// TIA Portal V15.1 export
// export: Created 2024-05-17T05:38:45.8173072Z, ExportSetting WithDefaults, DisplayName Totally Integrated Automation Portal, DisplayVersion V15.1 Update 5, DisplayName TIA Portal Openness, DisplayVersion V15.1 Update 5, DisplayName SINAMICS Startdrive Advanced, DisplayVersion V15.1, DisplayName G130, G150, S120, S150, SINAMICS MV, S210, DisplayVersion V15.1, DisplayName G110M, G120, G120C, G120D, G120P, DisplayVersion V15.1, DisplayName STEP 7 Professional, DisplayVersion V15.1 Update 5, DisplayName STEP 7 Safety, DisplayVersion V15.1, DisplayName WinCC Professional, DisplayVersion V15.1 Update 5, DisplayName SIMATIC Visualization Architect, DisplayVersion V15.1
FUNCTION_BLOCK "LGBGateLock-MGB-Maint"   // FB6628, FBD
TITLE = LGateLock-MGB / LGateLock-MGB-Maint
{ S7_Optimized_Access := 'TRUE' }
VERSION : 0.1
// =============================================================================
// This module is used for Euchner steered doorlock with 6 (lamp)pushbuttons and emergency stop
// Artikel 124573 MGB-L1HEB-PNA-R-124573
// Artikel 124575 MGB-L1HEB-PNA-L-124575
// 
// This module generates also a word containing all necessary information for HMI 
// Icon Animation, and a word with all information for HMI safety module 
// diagnostic screen. 
// =============================================================================
// stored: AutoNumber false, IsIECCheckEnabled false, IsRetainMemResEnabled false, MemoryReserve 100, SetENOAutomatically False, UDAEnableTagReadback false
   VAR_INPUT
      I_SafetyGateInput { ExternalAccessible := 'False'; ExternalVisible := 'False'; ExternalWritable := 'False'} : Bool;   // Input safety alarm (normally closed) / Input safety alarm (Summary door closed [T] and handle closed [R] - SK) / Input safety gate alarm (Summary door closed [T] and handle closed [R] - SK)
      I_Q { ExternalAccessible := 'False'; ExternalVisible := 'False'; ExternalWritable := 'False'} : Bool;   // Input safety alarm (normally closed) / Input Safety Alarm (normally closed) / Input Safety Logic Result Alarm (normally closed)
      I_EnableAlarm { ExternalAccessible := 'False'; ExternalVisible := 'False'; ExternalWritable := 'False'} : Bool := TRUE;   // Enable alarm from upper level
      I_StartPBInd { ExternalAccessible := 'False'; ExternalVisible := 'False'; ExternalWritable := 'False'} : Bool;   // Start PB indication
      I_AlarmResetPBInd { ExternalAccessible := 'False'; ExternalVisible := 'False'; ExternalWritable := 'False'} : Bool;   // Alarm reset PB indicatio / Alarm Reset PB Indication
      I_AccessStopReached { ExternalAccessible := 'False'; ExternalVisible := 'False'; ExternalWritable := 'False'} : Bool;   // Stop position reached for Request access / Access stop position reached
      I_CycleStopRequest { ExternalAccessible := 'False'; ExternalVisible := 'False'; ExternalWritable := 'False'} : Bool;   // Cycle stop request / Maintenance request
      I_CycleStopReached { ExternalAccessible := 'False'; ExternalVisible := 'False'; ExternalWritable := 'False'} : Bool;   // Cycle stop reached
      I_MaintRequest { ExternalAccessible := 'False'; ExternalVisible := 'False'; ExternalWritable := 'False'} : Bool;   // Cycle stop request / Maintenance request
      I_MaintReached { ExternalAccessible := 'False'; ExternalVisible := 'False'; ExternalWritable := 'False'} : Bool;   // Maintenance Position Reached
      I_SafetyCard_Pass_Out { ExternalAccessible := 'False'; ExternalVisible := 'False'; ExternalWritable := 'False'} : Bool;   // Passivation output
      I_SafetyCard_ACK_REQ { ExternalAccessible := 'False'; ExternalVisible := 'False'; ExternalWritable := 'False'} : Bool;   // ACK_REQ
      I_SafetyCard_ACK_DIAG { ExternalAccessible := 'False'; ExternalVisible := 'False'; ExternalWritable := 'False'} : Byte;   // ACK_DIAG
      "C_MGB-B" { ExternalAccessible := 'False'; ExternalVisible := 'False'; ExternalWritable := 'False'} : HW_SUBMODULE;   // Hw Config
      "C_MGB-EmergencySwitchStd" { ExternalAccessible := 'False'; ExternalVisible := 'False'; ExternalWritable := 'False'} : HW_SUBMODULE;   // Hw Config
      "C_MGB-L" { ExternalAccessible := 'False'; ExternalVisible := 'False'; ExternalWritable := 'False'} : HW_SUBMODULE;   // Hw Config
      "C_MBG-EnablingSwitchStd" { ExternalAccessible := 'False'; ExternalVisible := 'False'; ExternalWritable := 'False'} : HW_SUBMODULE;   // Hw Config
      "C_MBG-DIAG" { ExternalAccessible := 'False'; ExternalVisible := 'False'; ExternalWritable := 'False'} : HW_SUBMODULE;   // Hw Config
   END_VAR
   VAR_OUTPUT
      O_StartPB { ExternalAccessible := 'False'; ExternalVisible := 'False'; ExternalWritable := 'False'} : Bool;   // Pushbutton Start
      O_ResetAlarmPB { ExternalAccessible := 'False'; ExternalVisible := 'False'; ExternalWritable := 'False'} : Bool;   // Pushbutton Reset Alarm
      O_StopPB { ExternalAccessible := 'False'; ExternalVisible := 'False'; ExternalWritable := 'False'} : Bool;   // Pushbutton Stop (Delayed)
      O_EnablingSwitchPB { ExternalAccessible := 'False'; ExternalVisible := 'False'; ExternalWritable := 'False'} : Bool;   // Pushbutton Start / Pushbutton Enabling Switch
      "O_EnablingSwitch+PB" { ExternalAccessible := 'False'; ExternalVisible := 'False'; ExternalWritable := 'False'} : Bool;   // Pushbutton Start / Pushbutton Enabling Switch +
      "O_EnablingSwitch-PB" { ExternalAccessible := 'False'; ExternalVisible := 'False'; ExternalWritable := 'False'} : Bool;   // Pushbutton Start / Pushbutton Enabling Switch -
      O_MaintReq { ExternalAccessible := 'False'; ExternalVisible := 'False'; ExternalWritable := 'False'} : Bool;   // Switch Maintenance
      O_CycleStopReq { ExternalAccessible := 'False'; ExternalVisible := 'False'; ExternalWritable := 'False'} : Bool;   // Request for cycle stop / Request for Cycle Stop
      O_AccesStopReq { ExternalAccessible := 'False'; ExternalVisible := 'False'; ExternalWritable := 'False'} : Bool;   // Request for cycle stop / Request for Cycle Stop / Request for Acces Stop / Request for Access
      O_SafetyGateAlarm { ExternalAccessible := 'False'; ExternalVisible := 'False'; ExternalWritable := 'False'} : Bool;   // Alarm / Safety Alarm (Gate open) / Safety Gate Alarm
      O_EnablingSwitchAlarm { ExternalAccessible := 'False'; ExternalVisible := 'False'; ExternalWritable := 'False'} : Bool;   // Alarm / Enabling Switch Alarm (B) / Safety Gate Alarm
      O_SolenoidAlarm { ExternalAccessible := 'False'; ExternalVisible := 'False'; ExternalWritable := 'False'} : Bool;   // Summation Alarm A / Alarm / Alarm (C) / Solenoid Alarm
      O_AccessReqAlarm { ExternalAccessible := 'False'; ExternalVisible := 'False'; ExternalWritable := 'False'} : Bool;   // Alarm (C)
      O_MGBDiagWarning { ExternalAccessible := 'False'; ExternalVisible := 'False'; ExternalWritable := 'False'} : Bool;   // Summation Alarm C / Warning / Warning (D) / MGB diagnostic Warning
      O_AlarmABCondition { ExternalAccessible := 'False'; ExternalVisible := 'False'; ExternalWritable := 'False'} : Bool;   // Alarm AB Condition / Alarm AB condition
   END_VAR
   VAR_IN_OUT
      IO_Modes : "Modes";   // Modes
      H_HMI : "H_HMI";   // Animation
      "H_GateLock-MGB" : "H_GateLock-MGB-Maint";   // Animation
      C_AlarmHighSeverityA { ExternalAccessible := 'False'; ExternalVisible := 'False'; ExternalWritable := 'False'} : Bool := TRUE;   // Interlock alarm for Set direction / Alarm severity / Alarm severity A
      C_AlarmHighSeverityB { ExternalAccessible := 'False'; ExternalVisible := 'False'; ExternalWritable := 'False'} : Bool := False;   // Interlock alarm for Set direction / Alarm severity / Alarm severity B
      C_Warning { ExternalAccessible := 'False'; ExternalVisible := 'False'; ExternalWritable := 'False'} : Bool := False;   // Warning
   END_VAR
   VAR
      MGB { ExternalAccessible := 'False'; ExternalVisible := 'False'; ExternalWritable := 'False'} : "Euchner-MGB-Maint";   // UDT
      SafetyCard { ExternalAccessible := 'False'; ExternalVisible := 'False'; ExternalWritable := 'False'} : "SafetyCard";   // Safety Card UDT
      Pass_Out { ExternalAccessible := 'False'; ExternalVisible := 'False'; ExternalWritable := 'False'} : Bool;   // Acknowledgement request / Passivation output
      Ack_Req { ExternalAccessible := 'False'; ExternalVisible := 'False'; ExternalWritable := 'False'} : Bool;   // Acknowledgement request / Acknowledge Request
      Timeout_F_I_O { ExternalAccessible := 'False'; ExternalVisible := 'False'; ExternalWritable := 'False'} : Bool;   // Timeout detected by F-I/O
      ChannelFault_F_I_O { ExternalAccessible := 'False'; ExternalVisible := 'False'; ExternalWritable := 'False'} : Bool;   // F-I/O fault or channel fault detected by F-I/O
      CRCSeqError_F_I_O { ExternalAccessible := 'False'; ExternalVisible := 'False'; ExternalWritable := 'False'} : Bool;   // CRC error or sequence number error detected by F-I/O
      Timeout_F_Sys { ExternalAccessible := 'False'; ExternalVisible := 'False'; ExternalWritable := 'False'} : Bool;   // Timeout detected by F-System
      SeqError_F_Sys { ExternalAccessible := 'False'; ExternalVisible := 'False'; ExternalWritable := 'False'} : Bool;   // Sequence number error detected by F-system
      CRCError_F_Sys { ExternalAccessible := 'False'; ExternalVisible := 'False'; ExternalWritable := 'False'} : Bool;   // CRC error detected by F-system
      DelayStop { ExternalAccessible := 'False'; ExternalVisible := 'False'; ExternalWritable := 'False'} : Bool;   // Stop pushbutton delayed
      DelayMaint { ExternalAccessible := 'False'; ExternalVisible := 'False'; ExternalWritable := 'False'} : Bool;   // Maintenance pushbutton delayed
      SafetyGateAlarm { ExternalAccessible := 'False'; ExternalVisible := 'False'; ExternalWritable := 'False'} : Bool;   // Alarm / Safety Gate Alarm
      SafetyGateAlarmCond { ExternalAccessible := 'False'; ExternalVisible := 'False'; ExternalWritable := 'False'} : Bool;   // Alarm condition / Safety Gate Alarm condition
      EnablingSwitchAlarm { ExternalAccessible := 'False'; ExternalVisible := 'False'; ExternalWritable := 'False'} : Bool;   // Alarm / Safety Gate Alarm
      EnablingSwitchAlarmCond { ExternalAccessible := 'False'; ExternalVisible := 'False'; ExternalWritable := 'False'} : Bool;   // Alarm condition / Safety Gate Alarm condition
      SolenoidAlarm { ExternalAccessible := 'False'; ExternalVisible := 'False'; ExternalWritable := 'False'} : Bool;   // Alarm / Solenoid Alarm
      SolenoidAlarmCond { ExternalAccessible := 'False'; ExternalVisible := 'False'; ExternalWritable := 'False'} : Bool;   // Alarm condition / Solenoid Alarm condition
      AccessReqAlarm { ExternalAccessible := 'False'; ExternalVisible := 'False'; ExternalWritable := 'False'} : Bool;   // Alarm / Solenoid Alarm / Access Request Alarm
      DelayCheckGuardUnlocking { ExternalAccessible := 'False'; ExternalVisible := 'False'; ExternalWritable := 'False'} : Bool;   // Alarm / Alarm Delay to check guard locking / Alarm Delay to check guard unlocking
      AccessReqSel { ExternalAccessible := 'False'; ExternalVisible := 'False'; ExternalWritable := 'False'} : Bool;   // Request access memory / Request access selected
      AccessReq { ExternalAccessible := 'False'; ExternalVisible := 'False'; ExternalWritable := 'False'} : Bool;   // Request access memory / Request access
      NotAutoMem { ExternalAccessible := 'False'; ExternalVisible := 'False'; ExternalWritable := 'False'} : Bool;   // Pushbutton stop memory
      DelayTimerPbStop { ExternalAccessible := 'False'; ExternalVisible := 'False'; ExternalWritable := 'False'} : IEC_TIMER;   // Delay timer for Stop pushbutton
      DelayTimerSolenoidAlarm { ExternalAccessible := 'False'; ExternalVisible := 'False'; ExternalWritable := 'False'} : IEC_TIMER;   // Delay timer for solenoid Alarm
      DelayTimerMaintPb { ExternalAccessible := 'False'; ExternalVisible := 'False'; ExternalWritable := 'False'} : IEC_TIMER;   // Delay timer for maintenance pushbutton
      DelayOFFAutoMode { ExternalAccessible := 'False'; ExternalVisible := 'False'; ExternalWritable := 'False'} : IEC_TIMER;   // Delay OFF auto mode
      Edge { ExternalAccessible := 'False'; ExternalVisible := 'False'; ExternalWritable := 'False'} : Array[1..10] of Bool;   // Edges / Edge
      _ToggleReqAccess { ExternalAccessible := 'False'; ExternalVisible := 'False'; ExternalWritable := 'False'} : "LToggle";   // Toggle request access / Toggle access request
   END_VAR
   VAR_TEMP   // added for the SCL form of the ladder/FBD networks
      _w1 : Bool;
      _w2 : Bool;
   END_VAR
BEGIN

NETWORK
TITLE = **** 1 - Inputs **** Input Range - Output Range Euchner Safetylock
// Input Range - Output Range Euchner Safetylock
// Input range MGB-B
// Bit      7          6          5          4             3             2               1              0
// Byte 0   -          -          Stop       Cycle Stop    Maintenance   Request Access  Reset Alarm    Start

// Input range MGB-L
// Bit      7          6          5          4             3             2               1              0
// Byte 0   -          -          -          -             -             Door Locked     Handle Closed  Door Closed


// Output range MGB-B
// Bit      7          6          5          4             3             2               1              0
// Byte 0   -          -          -          Cycle Stop    Maintenance   Request Access  Reset Alarm    Start

// Output range MGB-L
// Bit      7          6          5          4             3             2               1              0
// Byte 0   -          -          -          -             -             -               -              Guard Locking



REGION Network 2: **** 1 - Inputs **** IN-Parameter reading and storing to local variables for MGB-B
   // IN-Parameter reading and storing to local variables for MGB-B
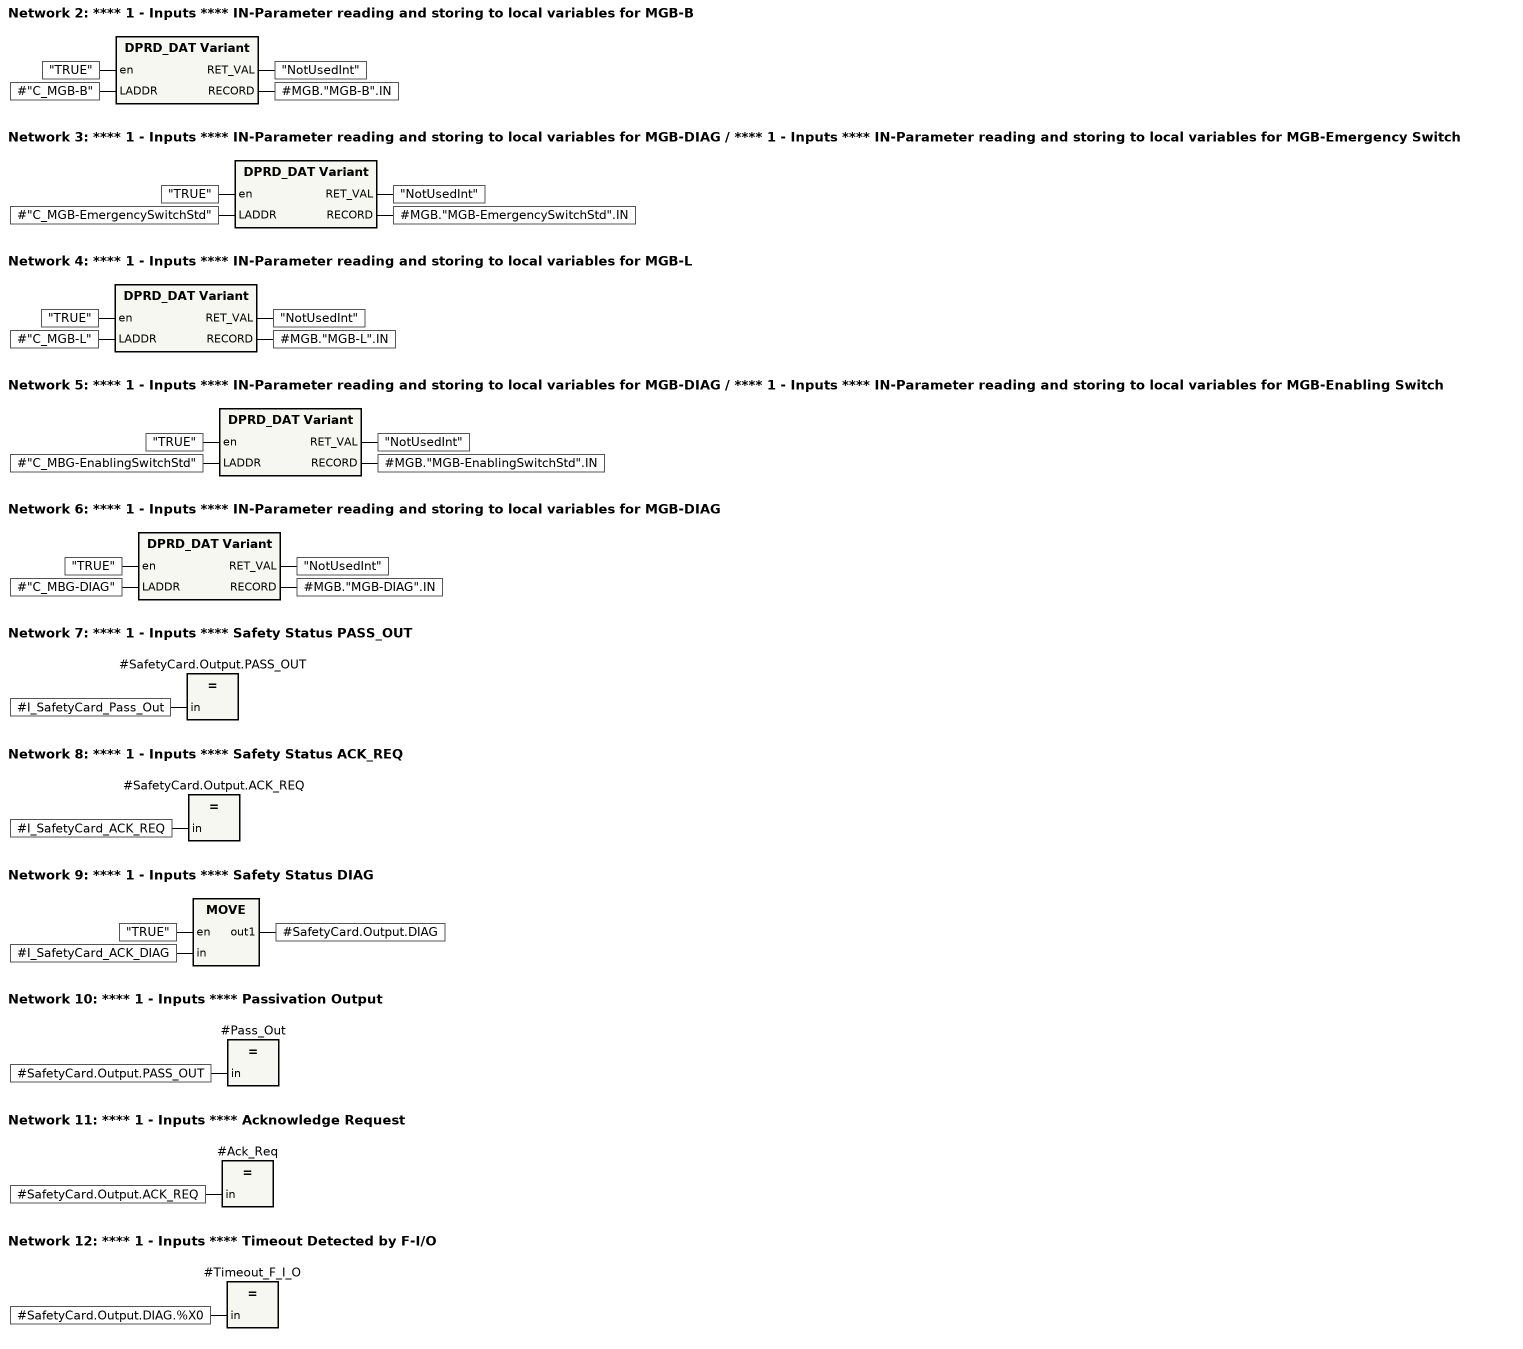
   IF "TRUE" THEN "NotUsedInt" := DPRD_DAT(LADDR := #"C_MGB-B", RECORD => #MGB."MGB-B".IN); END_IF;
END_REGION

REGION Network 3: **** 1 - Inputs **** IN-Parameter reading and storing to local variables for MGB-DIAG / **** 1 - Inputs **** IN-Parameter reading and storing to local variables for MGB-Emergency Switch
   // IN-Parameter reading and storing to local variables for MGB-DIAG / IN-Parameter reading and storing to local variables for MGB-Emergency Switch
   IF "TRUE" THEN
       "NotUsedInt" := DPRD_DAT(LADDR := #"C_MGB-EmergencySwitchStd", RECORD => #MGB."MGB-EmergencySwitchStd".IN);
   END_IF;
END_REGION

REGION Network 4: **** 1 - Inputs **** IN-Parameter reading and storing to local variables for MGB-L
   // IN-Parameter reading and storing to local variables for MGB-L
   IF "TRUE" THEN "NotUsedInt" := DPRD_DAT(LADDR := #"C_MGB-L", RECORD => #MGB."MGB-L".IN); END_IF;
END_REGION

REGION Network 5: **** 1 - Inputs **** IN-Parameter reading and storing to local variables for MGB-DIAG / **** 1 - Inputs **** IN-Parameter reading and storing to local variables for MGB-Enabling Switch
   // IN-Parameter reading and storing to local variables for MGB-DIAG / IN-Parameter reading and storing to local variables for MGB-Enabling Switch
   IF "TRUE" THEN
       "NotUsedInt" := DPRD_DAT(LADDR := #"C_MBG-EnablingSwitchStd", RECORD => #MGB."MGB-EnablingSwitchStd".IN);
   END_IF;
END_REGION

REGION Network 6: **** 1 - Inputs **** IN-Parameter reading and storing to local variables for MGB-DIAG
   // IN-Parameter reading and storing to local variables for MGB-DIAG
   IF "TRUE" THEN "NotUsedInt" := DPRD_DAT(LADDR := #"C_MBG-DIAG", RECORD => #MGB."MGB-DIAG".IN); END_IF;
END_REGION

REGION Network 7: **** 1 - Inputs **** Safety Status PASS_OUT
   // Safety Status PASS_OUT
   #SafetyCard.Output.PASS_OUT := #I_SafetyCard_Pass_Out;
END_REGION

REGION Network 8: **** 1 - Inputs **** Safety Status ACK_REQ
   // Safety Status ACK_REQ
   #SafetyCard.Output.ACK_REQ := #I_SafetyCard_ACK_REQ;
END_REGION

REGION Network 9: **** 1 - Inputs **** Safety Status DIAG
   // Safety Status DIAG
   IF "TRUE" THEN #SafetyCard.Output.DIAG := #I_SafetyCard_ACK_DIAG; END_IF;
END_REGION

REGION Network 10: **** 1 - Inputs **** Passivation Output
   // Passivation Output
   #Pass_Out := #SafetyCard.Output.PASS_OUT;
END_REGION

REGION Network 11: **** 1 - Inputs **** Acknowledge Request
   // Acknowledge Request
   #Ack_Req := #SafetyCard.Output.ACK_REQ;
END_REGION

REGION Network 12: **** 1 - Inputs **** Timeout Detected by F-I/O
   // ### Timeout Detected by F-I/O - must be checked
   #Timeout_F_I_O := #SafetyCard.Output.DIAG.%X0;
END_REGION

REGION Network 13: **** 1 - Inputs **** F-I/O fault or Channel Fault Detected by F-I/O
   // F-I/O fault or Channel Fault Detected by F-I/O
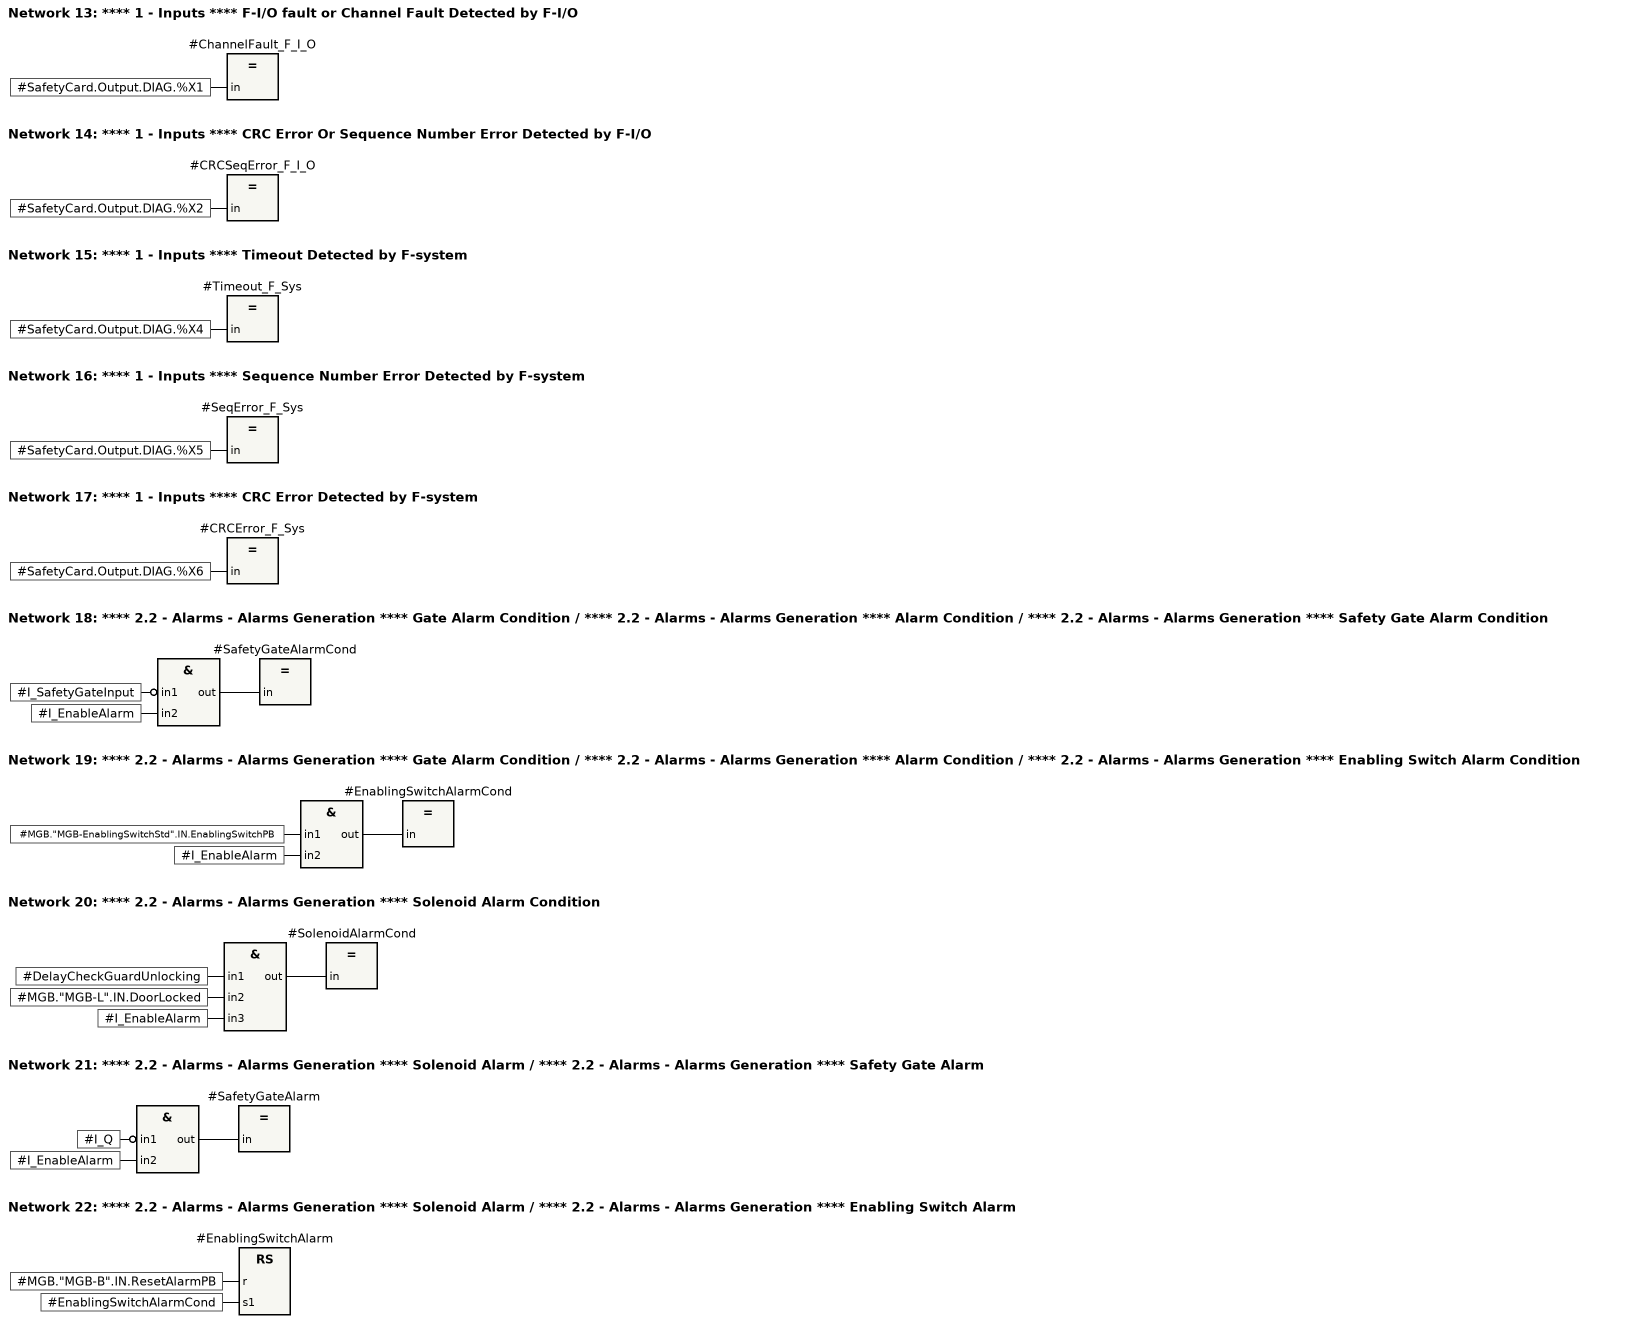
   #ChannelFault_F_I_O := #SafetyCard.Output.DIAG.%X1;
END_REGION

REGION Network 14: **** 1 - Inputs **** CRC Error Or Sequence Number Error Detected by F-I/O
   // CRC Error Or Sequence Number Error Detected by F-I/O
   #CRCSeqError_F_I_O := #SafetyCard.Output.DIAG.%X2;
END_REGION

REGION Network 15: **** 1 - Inputs **** Timeout Detected by F-system
   // Timeout Detected by F-system
   #Timeout_F_Sys := #SafetyCard.Output.DIAG.%X4;
END_REGION

REGION Network 16: **** 1 - Inputs **** Sequence Number Error Detected by F-system
   // Sequence Number Error Detected by F-system
   #SeqError_F_Sys := #SafetyCard.Output.DIAG.%X5;
END_REGION

REGION Network 17: **** 1 - Inputs **** CRC Error Detected by F-system
   // CRC Error Detected by F-system
   #CRCError_F_Sys := #SafetyCard.Output.DIAG.%X6;
END_REGION

REGION Network 18: **** 2.2 - Alarms - Alarms Generation **** Gate Alarm Condition / **** 2.2 - Alarms - Alarms Generation **** Alarm Condition / **** 2.2 - Alarms - Alarms Generation **** Safety Gate Alarm Condition
   // Condition of the Gate Alarm for the Normal Closed input / Condition of the Safety Alarm for the Normal Closed input
   #SafetyGateAlarmCond := NOT #I_SafetyGateInput AND #I_EnableAlarm;
END_REGION

REGION Network 19: **** 2.2 - Alarms - Alarms Generation **** Gate Alarm Condition / **** 2.2 - Alarms - Alarms Generation **** Alarm Condition / **** 2.2 - Alarms - Alarms Generation **** Enabling Switch Alarm Condition
   // Condition of the Gate Alarm for the Normal Closed input / Condition of the Safety Alarm for the Normal Closed input / Condition of the Enabling Switch actiavted alarm
   #EnablingSwitchAlarmCond := #MGB."MGB-EnablingSwitchStd".IN.EnablingSwitchPB AND #I_EnableAlarm;
END_REGION

REGION Network 20: **** 2.2 - Alarms - Alarms Generation **** Solenoid Alarm Condition
   // Condition of guardlocking on and solenoid not activated
   #SolenoidAlarmCond := #DelayCheckGuardUnlocking AND #MGB."MGB-L".IN.DoorLocked AND #I_EnableAlarm;
END_REGION

REGION Network 21: **** 2.2 - Alarms - Alarms Generation **** Solenoid Alarm / **** 2.2 - Alarms - Alarms Generation **** Safety Gate Alarm
   // Solenoid alarm / Condition of the Safety Alarm for the Normal Closed input
   #SafetyGateAlarm := NOT #I_Q AND #I_EnableAlarm;
END_REGION

REGION Network 22: **** 2.2 - Alarms - Alarms Generation **** Solenoid Alarm / **** 2.2 - Alarms - Alarms Generation **** Enabling Switch Alarm
   // Solenoid alarm / Enabling Switch alarm
   IF #MGB."MGB-B".IN.ResetAlarmPB THEN
       #EnablingSwitchAlarm := FALSE;   // RS flip-flop
   END_IF;
   IF #EnablingSwitchAlarmCond THEN #EnablingSwitchAlarm := TRUE; END_IF;
END_REGION

REGION Network 23: **** 2.2 - Alarms - Alarms Generation **** Solenoid Alarm
   // Solenoid alarm
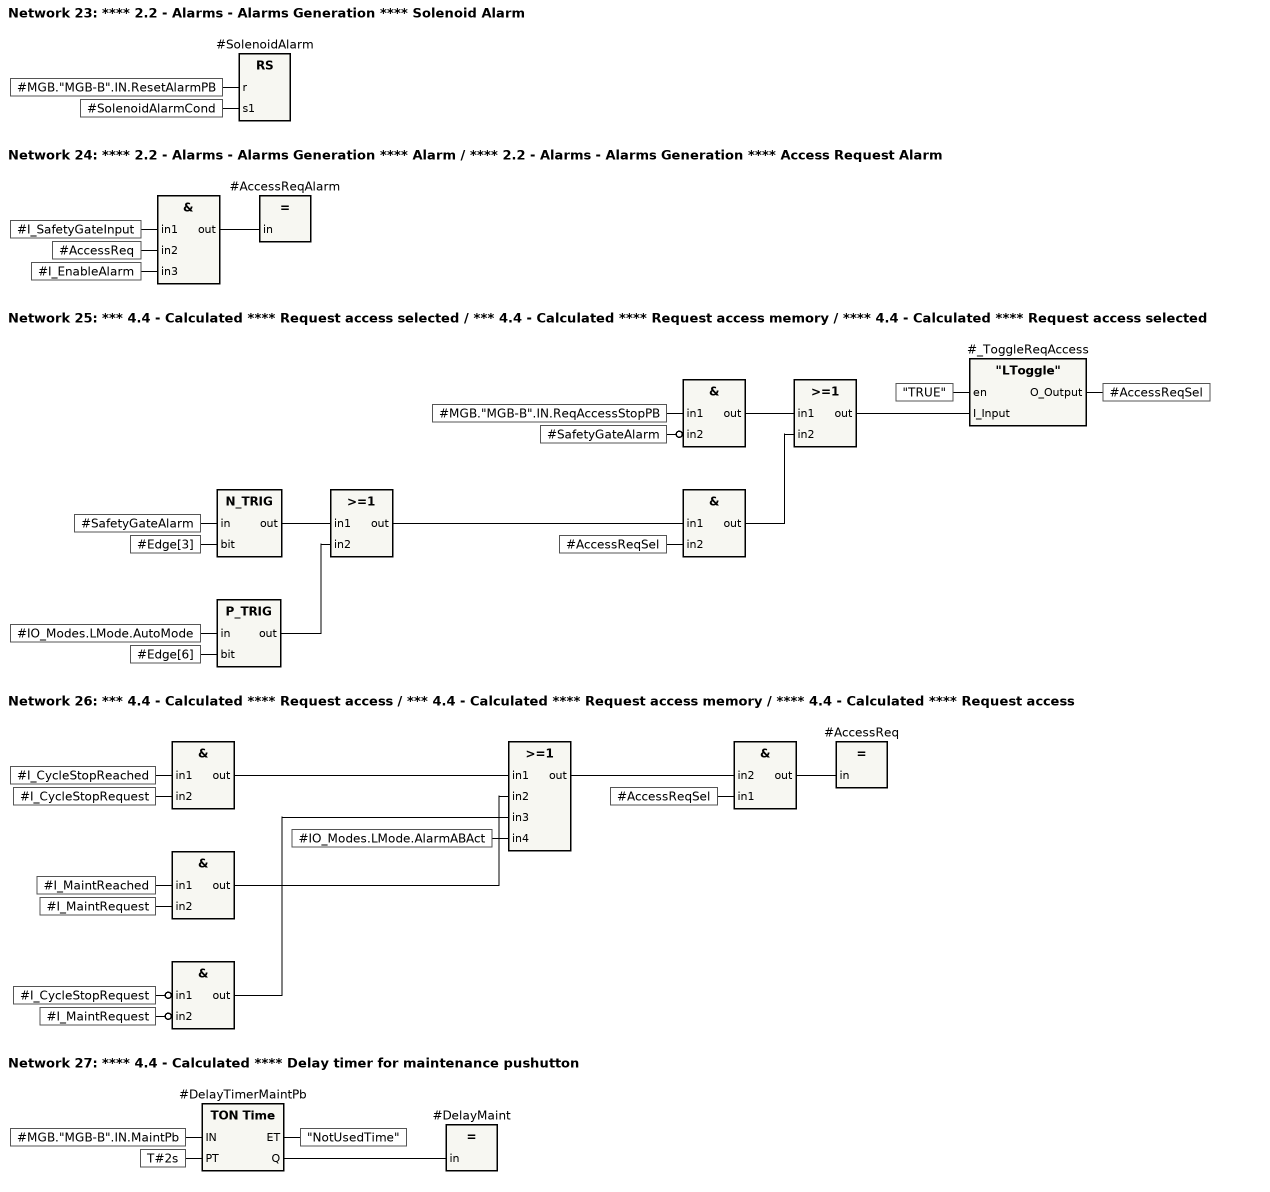
   IF #MGB."MGB-B".IN.ResetAlarmPB THEN
       #SolenoidAlarm := FALSE;   // RS flip-flop
   END_IF;
   IF #SolenoidAlarmCond THEN #SolenoidAlarm := TRUE; END_IF;
END_REGION

REGION Network 24: **** 2.2 - Alarms - Alarms Generation **** Alarm / **** 2.2 - Alarms - Alarms Generation **** Access Request Alarm
   // Creation of the Safety Alarm for the Normal Closed input / Alarm to notify that an access to the line is requested at the gate
   #AccessReqAlarm := #I_SafetyGateInput AND #AccessReq AND #I_EnableAlarm;
END_REGION

REGION Network 25: *** 4.4 - Calculated **** Request access selected / *** 4.4 - Calculated **** Request access memory / **** 4.4 - Calculated **** Request access selected
   // Request access selected / Request access memory
   #_w1 := NOT #SafetyGateAlarm AND #Edge[3];   // falling edge
   #Edge[3] := #SafetyGateAlarm;
   #_w2 := #IO_Modes.LMode.AutoMode AND NOT #Edge[6];   // rising edge
   #Edge[6] := #IO_Modes.LMode.AutoMode;
   IF "TRUE" THEN
       #_ToggleReqAccess(I_Input := (#MGB."MGB-B".IN.ReqAccessStopPB AND NOT #SafetyGateAlarm) OR ((#_w1 OR #_w2) AND #AccessReqSel),   // "LToggle"
                         O_Output => #AccessReqSel);
   END_IF;
END_REGION

REGION Network 26: *** 4.4 - Calculated **** Request access / *** 4.4 - Calculated **** Request access memory / **** 4.4 - Calculated **** Request access
   // Request access / Request access memory
   #AccessReq := ((#I_CycleStopReached AND #I_CycleStopRequest) OR (#I_MaintReached AND #I_MaintRequest) OR (NOT #I_CycleStopRequest AND NOT #I_MaintRequest) OR #IO_Modes.LMode.AlarmABAct) AND #AccessReqSel;
END_REGION

REGION Network 27: **** 4.4 - Calculated **** Delay timer for maintenance pushutton
   // Delay timer for maintenance pushutton
   #DelayTimerMaintPb.TON(IN := #MGB."MGB-B".IN.MaintPb, PT := T#2s, ET => "NotUsedTime");
   #DelayMaint := #DelayTimerMaintPb.Q;
END_REGION

REGION Network 28: *** 4.4 - Calculated **** Guard locking solenoid / **** 4.4 - Calculated **** Guard locking solenoid
   // Guard Locking Solenoid, Power to unlock (True = unlocked / False = locked) / Guard Locking Solenoid (True = locked / False = unlocked)
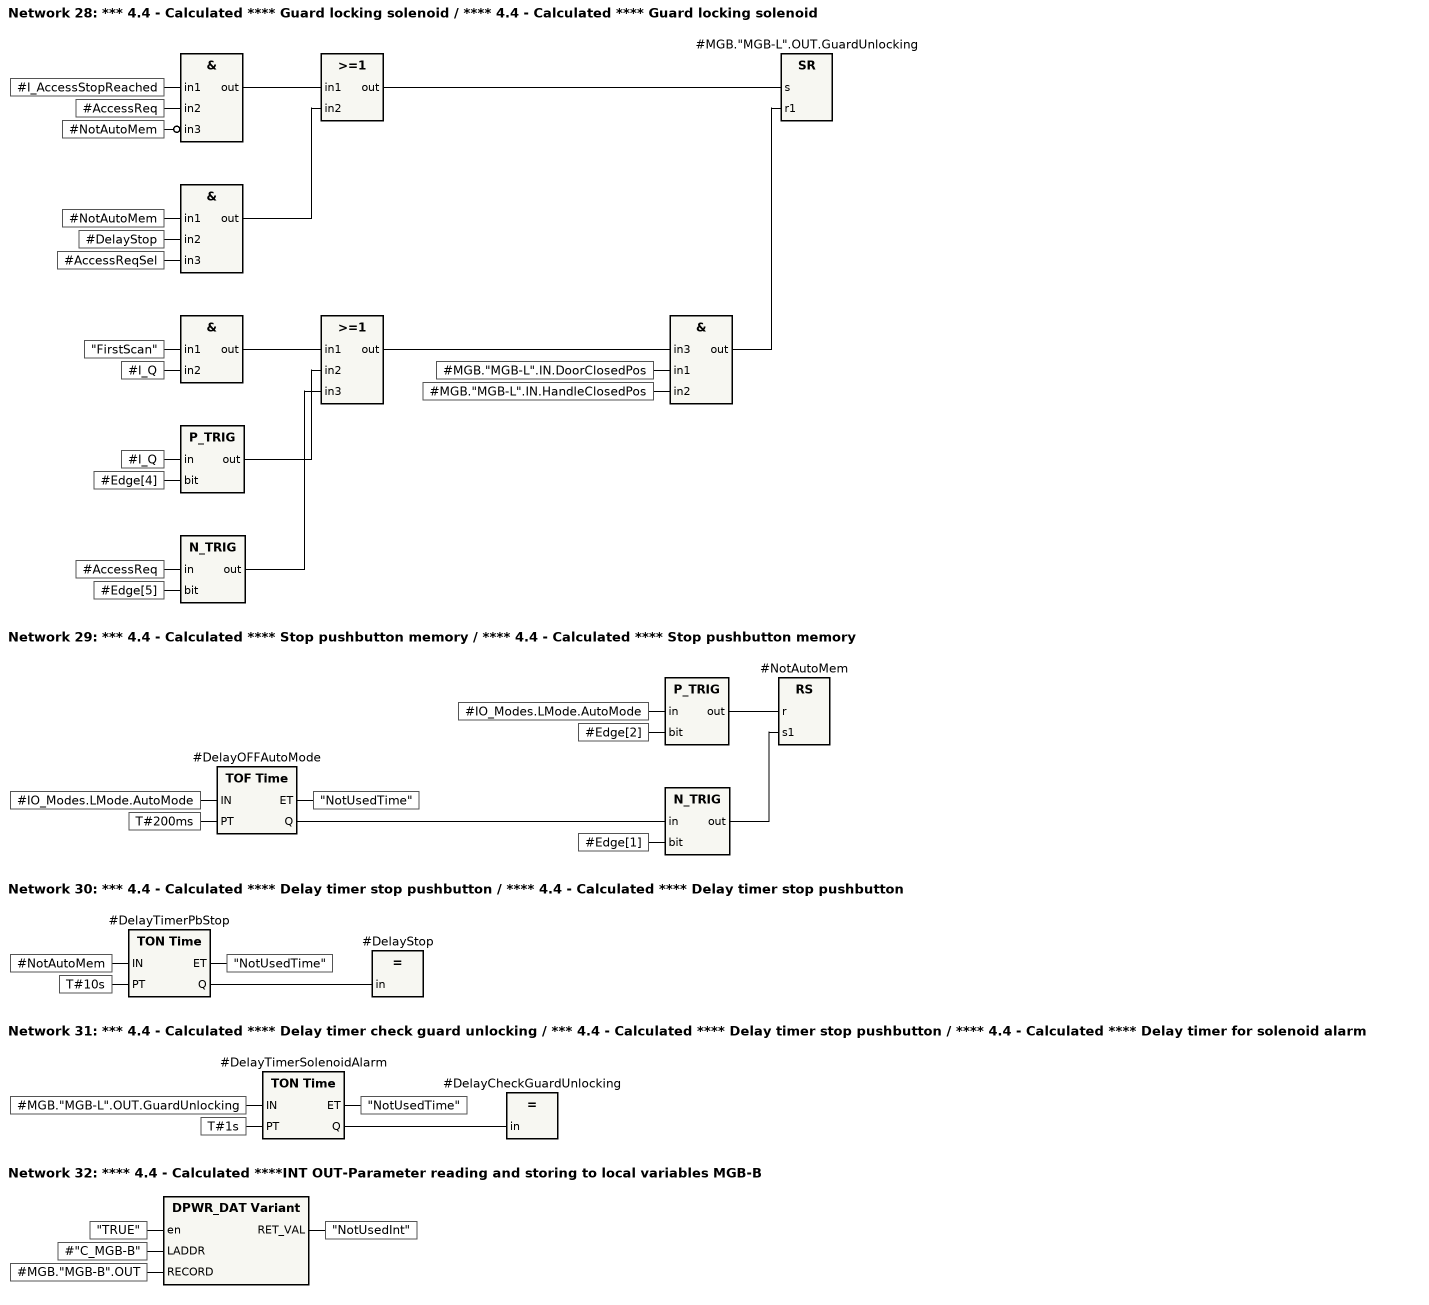
   #_w1 := #I_Q AND NOT #Edge[4];   // rising edge
   #Edge[4] := #I_Q;
   #_w2 := NOT #AccessReq AND #Edge[5];   // falling edge
   #Edge[5] := #AccessReq;
   IF (#I_AccessStopReached AND #AccessReq AND NOT #NotAutoMem) OR (#NotAutoMem AND #DelayStop AND #AccessReqSel) THEN
       #MGB."MGB-L".OUT.GuardUnlocking := TRUE;   // SR flip-flop
   END_IF;
   IF (("FirstScan" AND #I_Q) OR #_w1 OR #_w2) AND #MGB."MGB-L".IN.DoorClosedPos AND #MGB."MGB-L".IN.HandleClosedPos THEN
       #MGB."MGB-L".OUT.GuardUnlocking := FALSE;
   END_IF;
END_REGION

REGION Network 29: *** 4.4 - Calculated **** Stop pushbutton memory / **** 4.4 - Calculated **** Stop pushbutton memory
   // Stop pushbutton memory
   #_w1 := #IO_Modes.LMode.AutoMode AND NOT #Edge[2];   // rising edge
   #Edge[2] := #IO_Modes.LMode.AutoMode;
   #DelayOFFAutoMode.TOF(IN := #IO_Modes.LMode.AutoMode, PT := T#200ms, ET => "NotUsedTime");
   #_w2 := NOT #DelayOFFAutoMode.Q AND #Edge[1];   // falling edge
   #Edge[1] := #DelayOFFAutoMode.Q;
   IF #_w1 THEN
       #NotAutoMem := FALSE;   // RS flip-flop
   END_IF;
   IF #_w2 THEN #NotAutoMem := TRUE; END_IF;
END_REGION

REGION Network 30: *** 4.4 - Calculated **** Delay timer stop pushbutton / **** 4.4 - Calculated **** Delay timer stop pushbutton
   // Delay for Stop pushbutton
   #DelayTimerPbStop.TON(IN := #NotAutoMem, PT := T#10s, ET => "NotUsedTime");
   #DelayStop := #DelayTimerPbStop.Q;
END_REGION

REGION Network 31: *** 4.4 - Calculated **** Delay timer check guard unlocking / *** 4.4 - Calculated **** Delay timer stop pushbutton / **** 4.4 - Calculated **** Delay timer for solenoid alarm
   // Delay for checking of guard unlocking / Delay for Stop pushbutton / Delay timer for solenoid alarm
   #DelayTimerSolenoidAlarm.TON(IN := #MGB."MGB-L".OUT.GuardUnlocking, PT := T#1s, ET => "NotUsedTime");
   #DelayCheckGuardUnlocking := #DelayTimerSolenoidAlarm.Q;
END_REGION

REGION Network 32: **** 4.4 - Calculated ****INT OUT-Parameter reading and storing to local variables MGB-B
   // INT OUT-Parameter reading and storing to local variables MGB-B
   IF "TRUE" THEN "NotUsedInt" := DPWR_DAT(LADDR := #"C_MGB-B", RECORD := #MGB."MGB-B".OUT); END_IF;
END_REGION

REGION Network 33: **** 4.4 - Calculated ****INT OUT-Parameter reading and storing to local variables MGB Diag / **** 4.4 - Calculated ****INT OUT-Parameter reading and storing to local variables MGB-Emergency Switch
   // INT OUT-Parameter reading and storing to local variables MGB Diag / INT OUT-Parameter reading and storing to local variables MGB-Emergency Switch
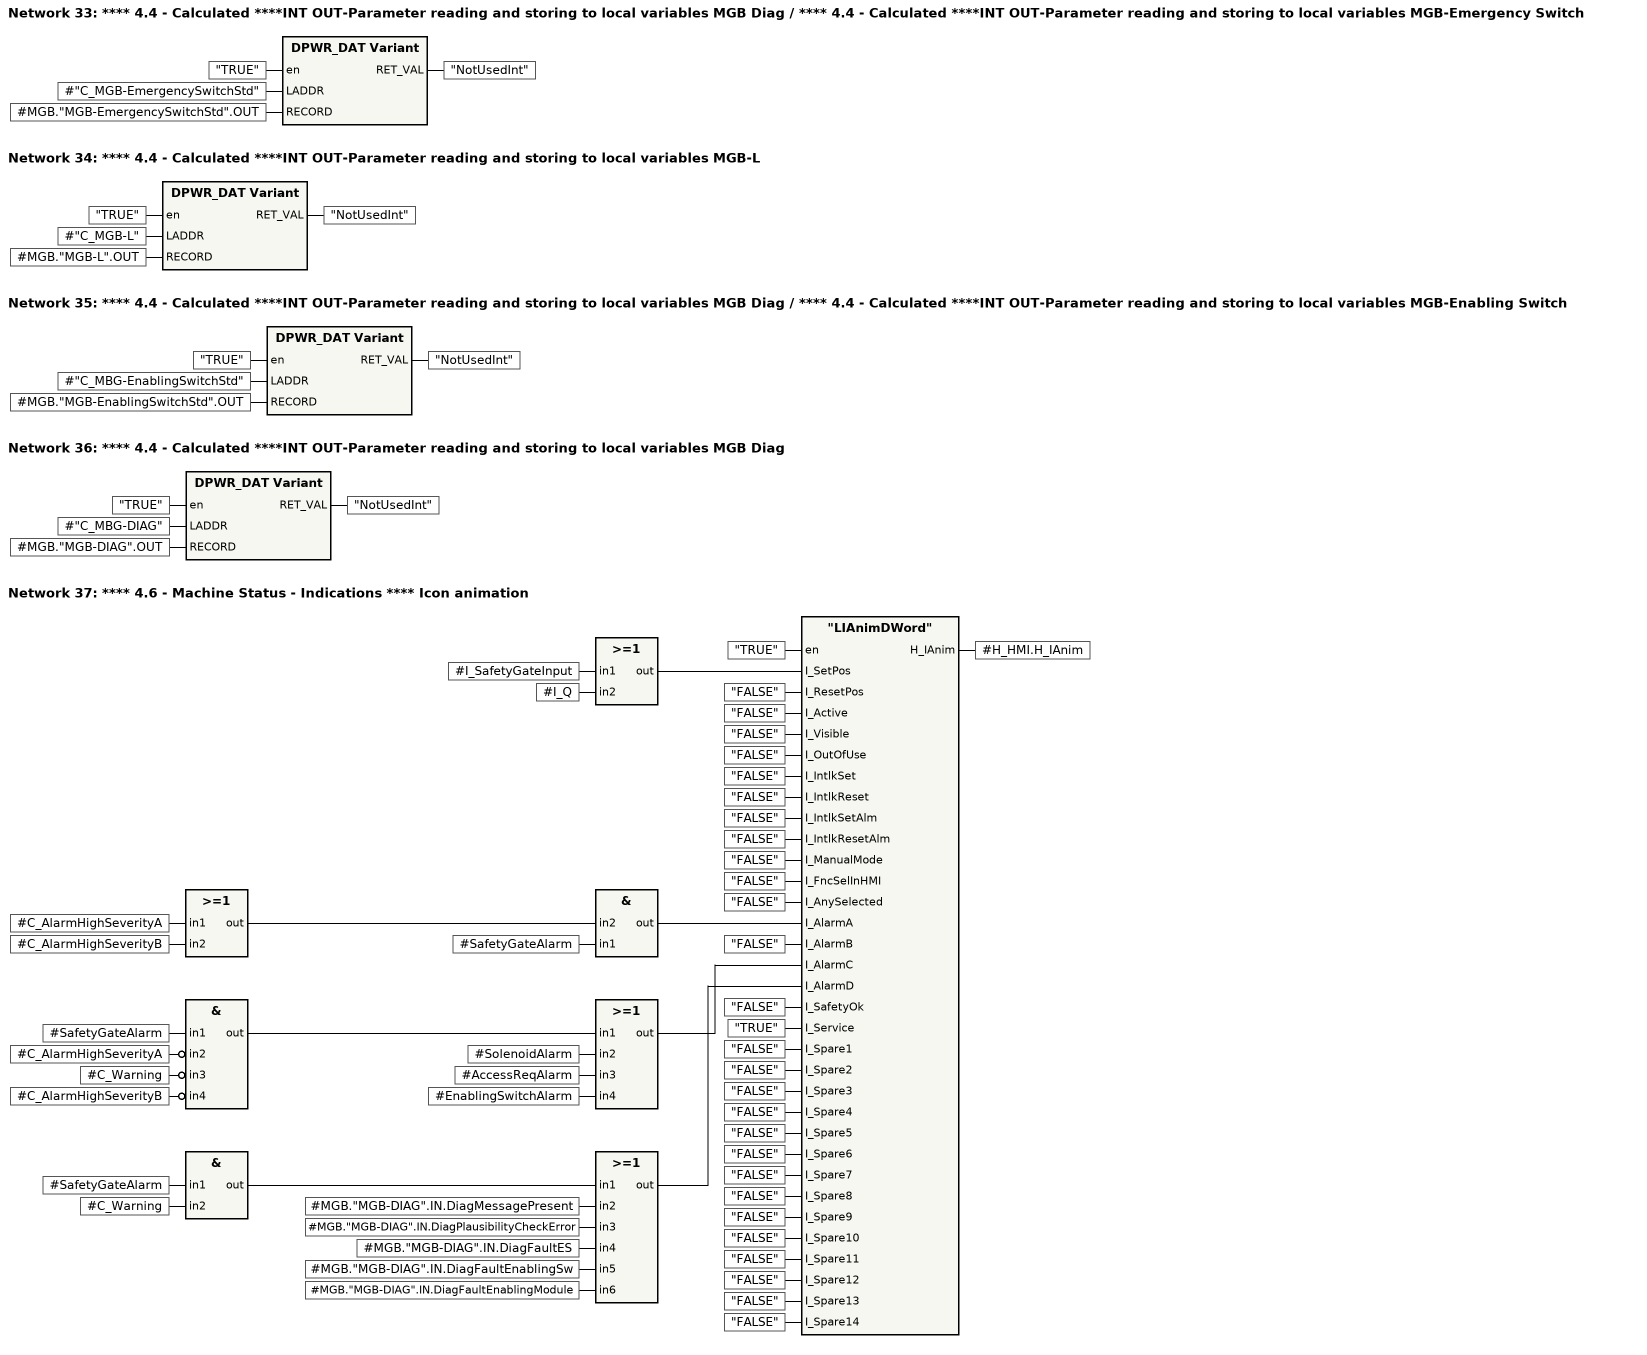
   IF "TRUE" THEN
       "NotUsedInt" := DPWR_DAT(LADDR := #"C_MGB-EmergencySwitchStd", RECORD := #MGB."MGB-EmergencySwitchStd".OUT);
   END_IF;
END_REGION

REGION Network 34: **** 4.4 - Calculated ****INT OUT-Parameter reading and storing to local variables MGB-L
   // INT OUT-Parameter reading and storing to local variables MGB-L
   IF "TRUE" THEN "NotUsedInt" := DPWR_DAT(LADDR := #"C_MGB-L", RECORD := #MGB."MGB-L".OUT); END_IF;
END_REGION

REGION Network 35: **** 4.4 - Calculated ****INT OUT-Parameter reading and storing to local variables MGB Diag / **** 4.4 - Calculated ****INT OUT-Parameter reading and storing to local variables MGB-Enabling Switch
   // INT OUT-Parameter reading and storing to local variables MGB Diag / INT OUT-Parameter reading and storing to local variables MGB-Enabling Switch
   IF "TRUE" THEN
       "NotUsedInt" := DPWR_DAT(LADDR := #"C_MBG-EnablingSwitchStd", RECORD := #MGB."MGB-EnablingSwitchStd".OUT);
   END_IF;
END_REGION

REGION Network 36: **** 4.4 - Calculated ****INT OUT-Parameter reading and storing to local variables MGB Diag
   // INT OUT-Parameter reading and storing to local variables MGB Diag
   IF "TRUE" THEN "NotUsedInt" := DPWR_DAT(LADDR := #"C_MBG-DIAG", RECORD := #MGB."MGB-DIAG".OUT); END_IF;
END_REGION

REGION Network 37: **** 4.6 - Machine Status - Indications **** Icon animation
   // Icon Animation
   IF "TRUE" THEN
       "LIAnimDWord"(I_SetPos := #I_SafetyGateInput OR #I_Q,
                     I_ResetPos := "FALSE",
                     I_Active := "FALSE",
                     I_Visible := "FALSE",
                     I_OutOfUse := "FALSE",
                     I_IntlkSet := "FALSE",
                     I_IntlkReset := "FALSE",
                     I_IntlkSetAlm := "FALSE",
                     I_IntlkResetAlm := "FALSE",
                     I_ManualMode := "FALSE",
                     I_FncSelInHMI := "FALSE",
                     I_AnySelected := "FALSE",
                     I_AlarmA := (#C_AlarmHighSeverityA OR #C_AlarmHighSeverityB) AND #SafetyGateAlarm,
                     I_AlarmB := "FALSE",
                     I_AlarmC := (#SafetyGateAlarm AND NOT #C_AlarmHighSeverityA AND NOT #C_Warning AND NOT #C_AlarmHighSeverityB) OR #SolenoidAlarm OR #AccessReqAlarm OR #EnablingSwitchAlarm,
                     I_AlarmD := (#SafetyGateAlarm AND #C_Warning) OR #MGB."MGB-DIAG".IN.DiagMessagePresent OR #MGB."MGB-DIAG".IN.DiagPlausibilityCheckError OR #MGB."MGB-DIAG".IN.DiagFaultES OR #MGB."MGB-DIAG".IN.DiagFaultEnablingSw OR #MGB."MGB-DIAG".IN.DiagFaultEnablingModule,
                     I_SafetyOk := "FALSE",
                     I_Service := "TRUE",
                     I_Spare1 := "FALSE",
                     I_Spare2 := "FALSE",
                     I_Spare3 := "FALSE",
                     I_Spare4 := "FALSE",
                     I_Spare5 := "FALSE",
                     I_Spare6 := "FALSE",
                     I_Spare7 := "FALSE",
                     I_Spare8 := "FALSE",
                     I_Spare9 := "FALSE",
                     I_Spare10 := "FALSE",
                     I_Spare11 := "FALSE",
                     I_Spare12 := "FALSE",
                     I_Spare13 := "FALSE",
                     I_Spare14 := "FALSE",
                     H_IAnim => #H_HMI.H_IAnim);
   END_IF;
END_REGION

REGION Network 38: **** 4.6 - Machine Status - Indications **** Animation
   // Animation
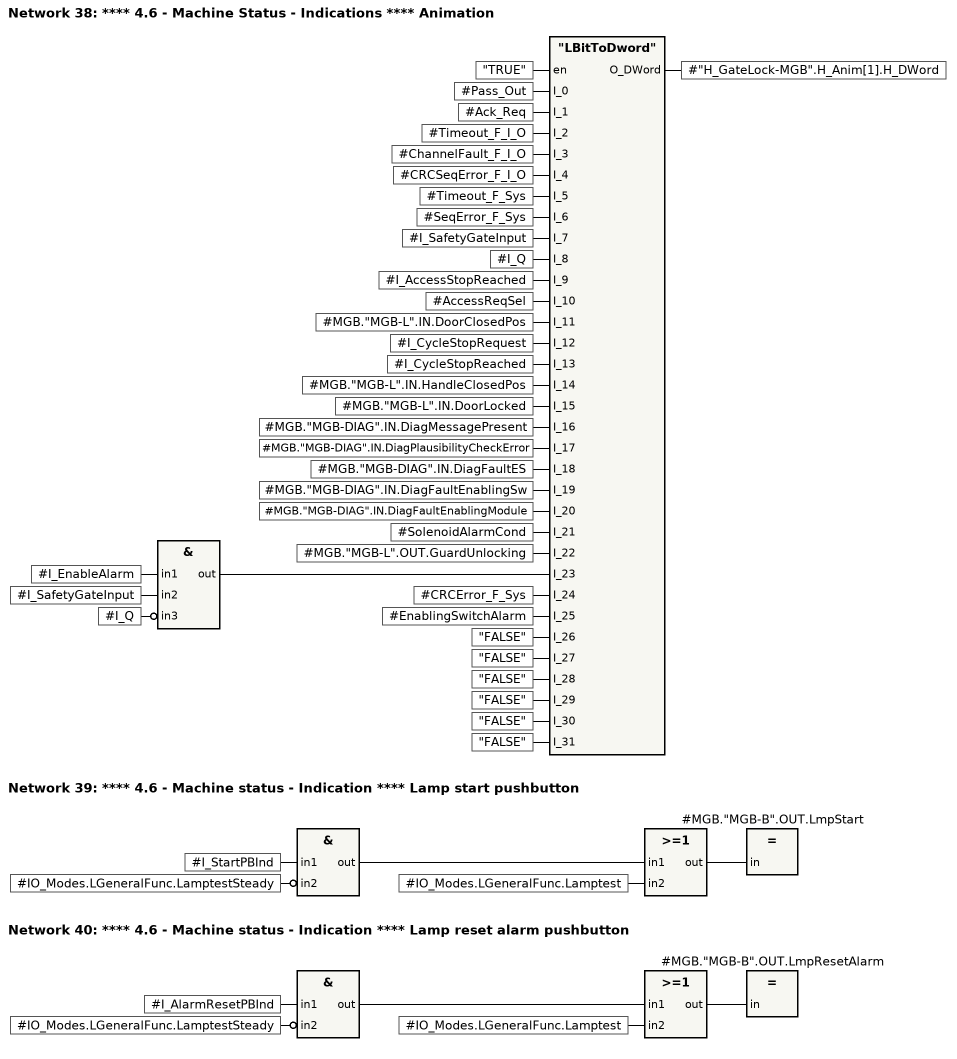
   IF "TRUE" THEN
       "LBitToDword"(I_0 := #Pass_Out,
                     I_1 := #Ack_Req,
                     I_2 := #Timeout_F_I_O,
                     I_3 := #ChannelFault_F_I_O,
                     I_4 := #CRCSeqError_F_I_O,
                     I_5 := #Timeout_F_Sys,
                     I_6 := #SeqError_F_Sys,
                     I_7 := #I_SafetyGateInput,
                     I_8 := #I_Q,
                     I_9 := #I_AccessStopReached,
                     I_10 := #AccessReqSel,
                     I_11 := #MGB."MGB-L".IN.DoorClosedPos,
                     I_12 := #I_CycleStopRequest,
                     I_13 := #I_CycleStopReached,
                     I_14 := #MGB."MGB-L".IN.HandleClosedPos,
                     I_15 := #MGB."MGB-L".IN.DoorLocked,
                     I_16 := #MGB."MGB-DIAG".IN.DiagMessagePresent,
                     I_17 := #MGB."MGB-DIAG".IN.DiagPlausibilityCheckError,
                     I_18 := #MGB."MGB-DIAG".IN.DiagFaultES,
                     I_19 := #MGB."MGB-DIAG".IN.DiagFaultEnablingSw,
                     I_20 := #MGB."MGB-DIAG".IN.DiagFaultEnablingModule,
                     I_21 := #SolenoidAlarmCond,
                     I_22 := #MGB."MGB-L".OUT.GuardUnlocking,
                     I_23 := #I_EnableAlarm AND #I_SafetyGateInput AND NOT #I_Q,
                     I_24 := #CRCError_F_Sys,
                     I_25 := #EnablingSwitchAlarm,
                     I_26 := "FALSE",
                     I_27 := "FALSE",
                     I_28 := "FALSE",
                     I_29 := "FALSE",
                     I_30 := "FALSE",
                     I_31 := "FALSE",
                     O_DWord => #"H_GateLock-MGB".H_Anim[1].H_DWord);
   END_IF;
END_REGION

REGION Network 39: **** 4.6 - Machine status - Indication **** Lamp start pushbutton
   // Start PB indication
   #MGB."MGB-B".OUT.LmpStart := (#I_StartPBInd AND NOT #IO_Modes.LGeneralFunc.LamptestSteady) OR #IO_Modes.LGeneralFunc.Lamptest;
END_REGION

REGION Network 40: **** 4.6 - Machine status - Indication **** Lamp reset alarm pushbutton
   // Reset Alarm PB indication / Alarm Reset PB indication
   #MGB."MGB-B".OUT.LmpResetAlarm := (#I_AlarmResetPBInd AND NOT #IO_Modes.LGeneralFunc.LamptestSteady) OR #IO_Modes.LGeneralFunc.Lamptest;
END_REGION

REGION Network 41: **** 4.6 - Machine status - Indication **** Lamp request access pushbutton
   // Request Acces PB indication
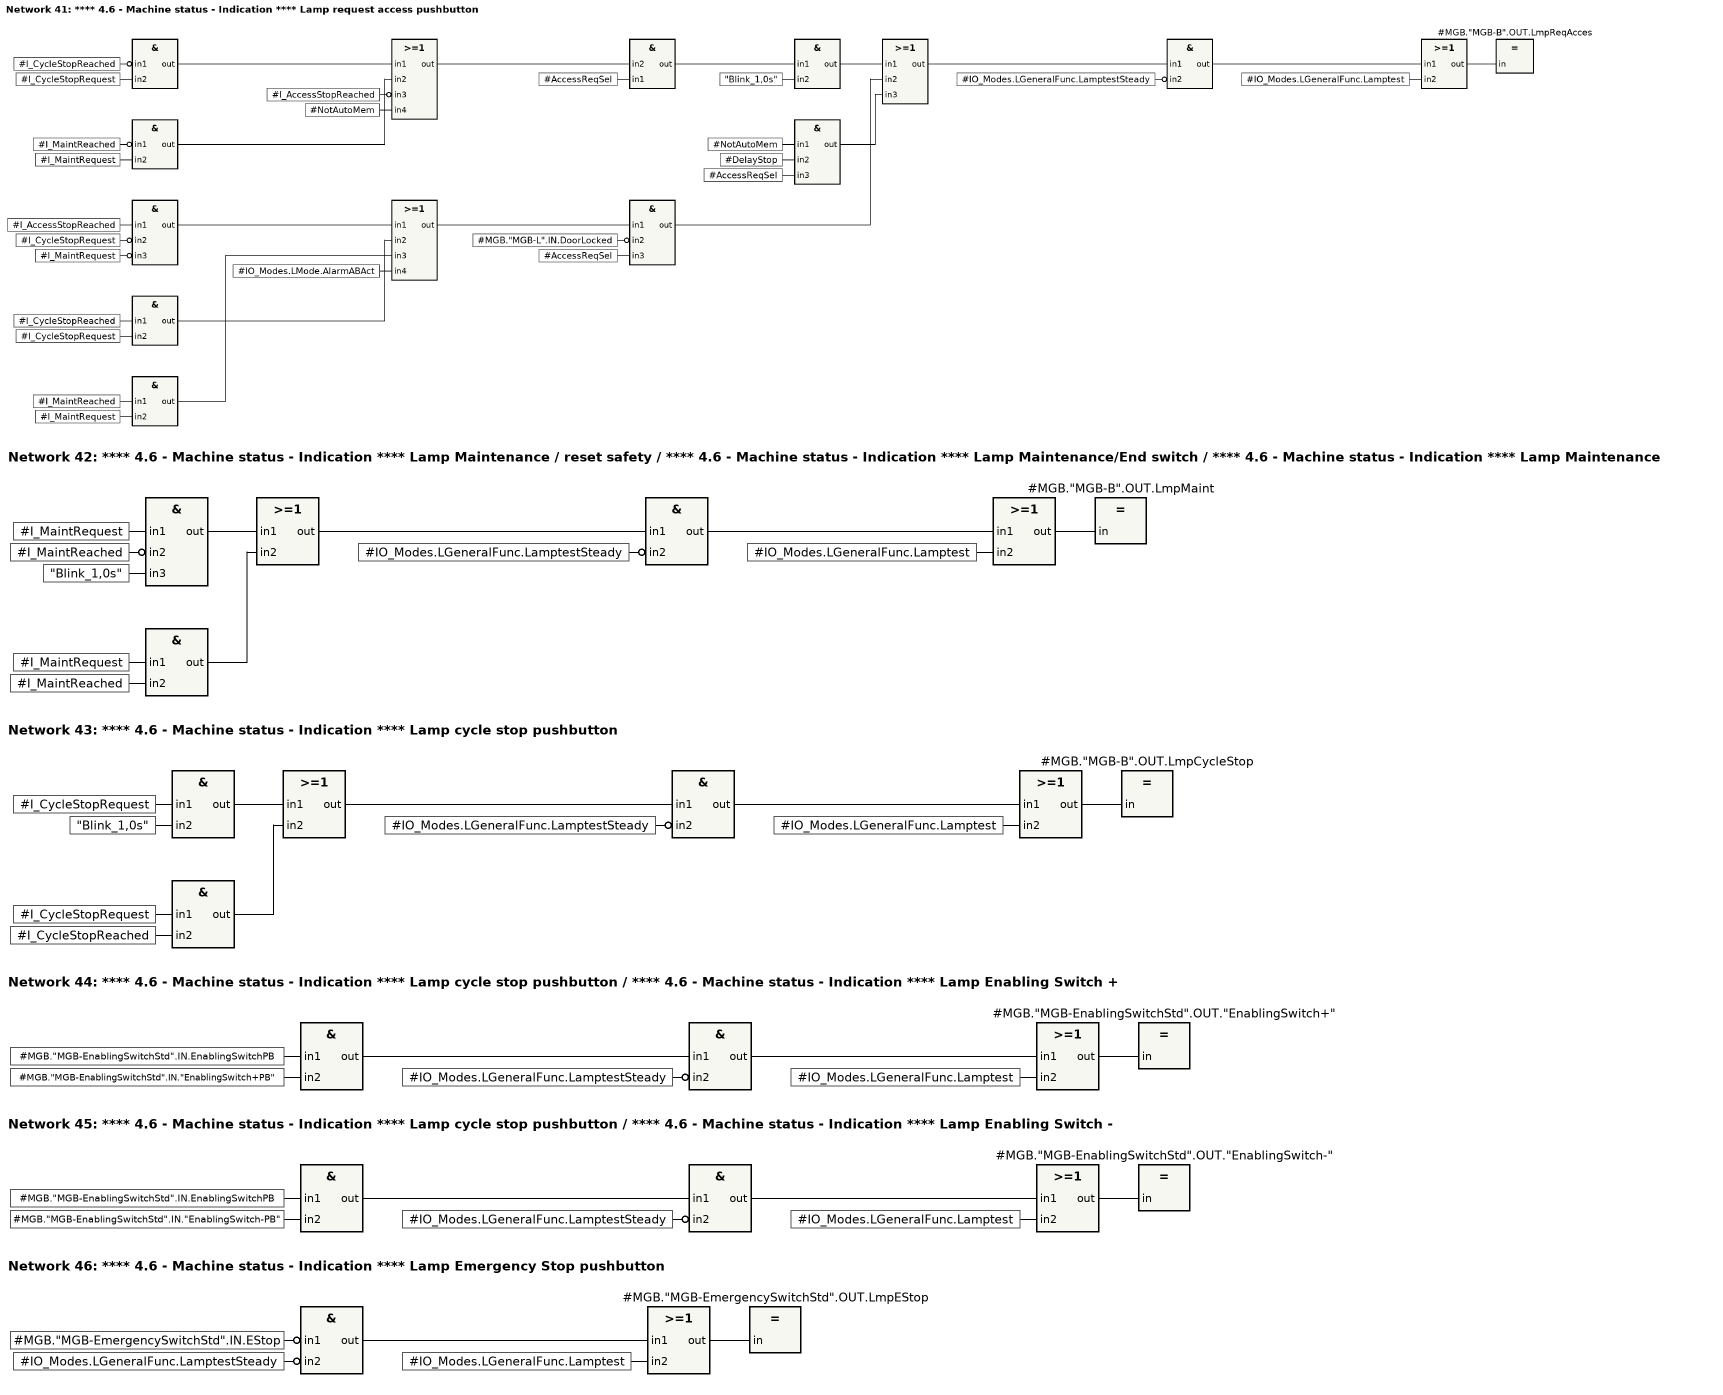
   #MGB."MGB-B".OUT.LmpReqAcces := (((((NOT #I_CycleStopReached AND #I_CycleStopRequest) OR (NOT #I_MaintReached AND #I_MaintRequest) OR NOT #I_AccessStopReached OR #NotAutoMem) AND #AccessReqSel AND "Blink_1,0s") OR (((#I_AccessStopReached AND NOT #I_CycleStopRequest AND NOT #I_MaintRequest) OR (#I_CycleStopReached AND #I_CycleStopRequest) OR (#I_MaintReached AND #I_MaintRequest) OR #IO_Modes.LMode.AlarmABAct) AND NOT #MGB."MGB-L".IN.DoorLocked AND #AccessReqSel) OR (#NotAutoMem AND #DelayStop AND #AccessReqSel)) AND NOT #IO_Modes.LGeneralFunc.LamptestSteady) OR #IO_Modes.LGeneralFunc.Lamptest;
END_REGION

REGION Network 42: **** 4.6 - Machine status - Indication **** Lamp Maintenance / reset safety / **** 4.6 - Machine status - Indication **** Lamp Maintenance/End switch / **** 4.6 - Machine status - Indication **** Lamp Maintenance
   // Maintenance/End SW indication / Maintenance Pb indication
   #MGB."MGB-B".OUT.LmpMaint := (((#I_MaintRequest AND NOT #I_MaintReached AND "Blink_1,0s") OR (#I_MaintRequest AND #I_MaintReached)) AND NOT #IO_Modes.LGeneralFunc.LamptestSteady) OR #IO_Modes.LGeneralFunc.Lamptest;
END_REGION

REGION Network 43: **** 4.6 - Machine status - Indication **** Lamp cycle stop pushbutton
   // Cycle Stop PB indication
   #MGB."MGB-B".OUT.LmpCycleStop := (((#I_CycleStopRequest AND "Blink_1,0s") OR (#I_CycleStopRequest AND #I_CycleStopReached)) AND NOT #IO_Modes.LGeneralFunc.LamptestSteady) OR #IO_Modes.LGeneralFunc.Lamptest;
END_REGION

REGION Network 44: **** 4.6 - Machine status - Indication **** Lamp cycle stop pushbutton / **** 4.6 - Machine status - Indication **** Lamp Enabling Switch +
   // Cycle Stop PB indication / Enabling Switch PB + indication
   #MGB."MGB-EnablingSwitchStd".OUT."EnablingSwitch+" := (#MGB."MGB-EnablingSwitchStd".IN.EnablingSwitchPB AND #MGB."MGB-EnablingSwitchStd".IN."EnablingSwitch+PB" AND NOT #IO_Modes.LGeneralFunc.LamptestSteady) OR #IO_Modes.LGeneralFunc.Lamptest;
END_REGION

REGION Network 45: **** 4.6 - Machine status - Indication **** Lamp cycle stop pushbutton / **** 4.6 - Machine status - Indication **** Lamp Enabling Switch -
   // Cycle Stop PB indication / Enabling Switch PB - indication
   #MGB."MGB-EnablingSwitchStd".OUT."EnablingSwitch-" := (#MGB."MGB-EnablingSwitchStd".IN.EnablingSwitchPB AND #MGB."MGB-EnablingSwitchStd".IN."EnablingSwitch-PB" AND NOT #IO_Modes.LGeneralFunc.LamptestSteady) OR #IO_Modes.LGeneralFunc.Lamptest;
END_REGION

REGION Network 46: **** 4.6 - Machine status - Indication **** Lamp Emergency Stop pushbutton
   #MGB."MGB-EmergencySwitchStd".OUT.LmpEStop := (NOT #MGB."MGB-EmergencySwitchStd".IN.EStop AND NOT #IO_Modes.LGeneralFunc.LamptestSteady) OR #IO_Modes.LGeneralFunc.Lamptest;
END_REGION

REGION Network 47: **** 5.2 - Equations - Equations **** Diagnostic Message Acknowledge / **** 5.2 - Equations - Equations **** High Speed Manual / **** 5.2 - Equations - Equations **** Diagnostic message Acknowlegde
   // Diagnostic Message Acknowledge / Cmd summary high speed in manual / Diagnostic message Acknowlegde
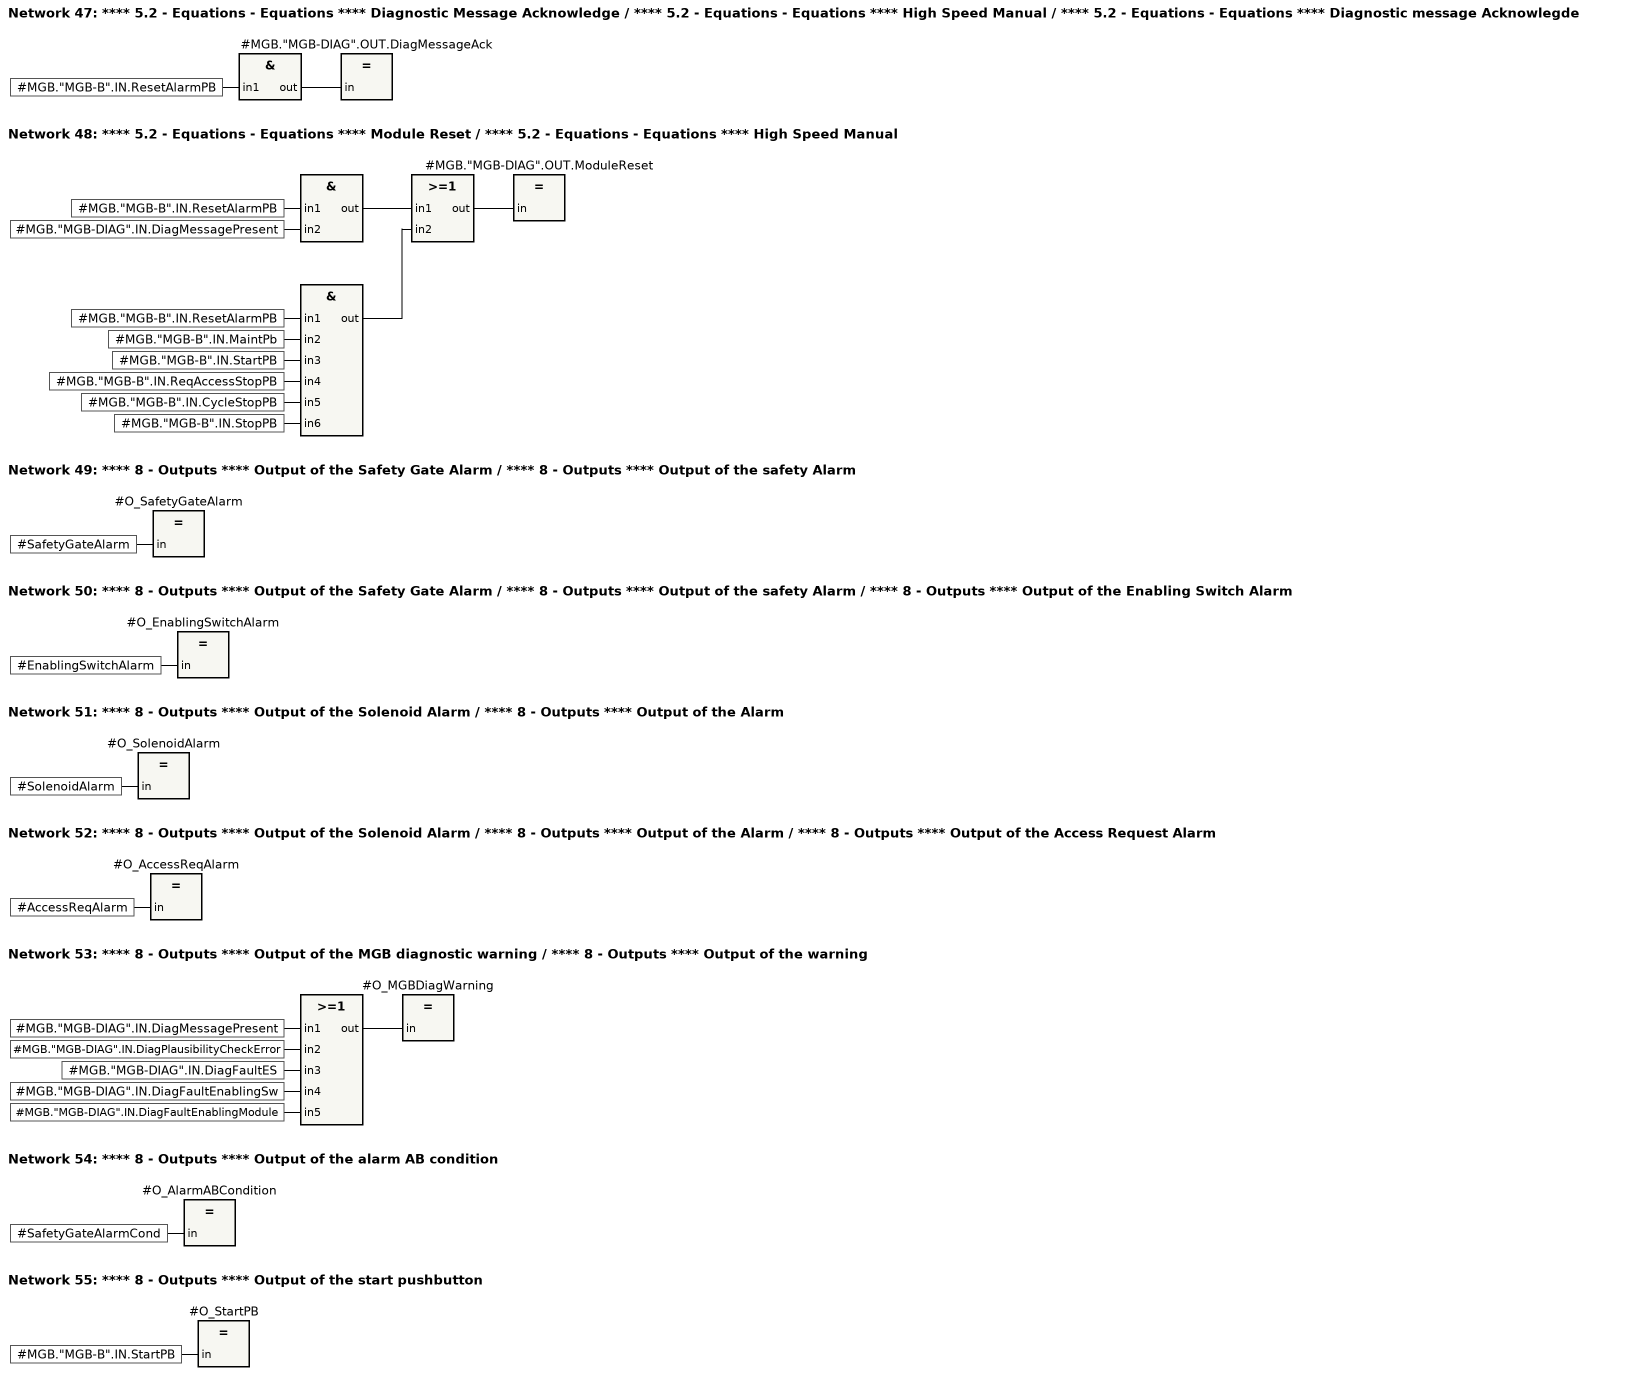
   #MGB."MGB-DIAG".OUT.DiagMessageAck := #MGB."MGB-B".IN.ResetAlarmPB;
END_REGION

REGION Network 48: **** 5.2 - Equations - Equations **** Module Reset / **** 5.2 - Equations - Equations **** High Speed Manual
   // Module Reset / Cmd summary high speed in manual
   #MGB."MGB-DIAG".OUT.ModuleReset := (#MGB."MGB-B".IN.ResetAlarmPB AND #MGB."MGB-DIAG".IN.DiagMessagePresent) OR (#MGB."MGB-B".IN.ResetAlarmPB AND #MGB."MGB-B".IN.MaintPb AND #MGB."MGB-B".IN.StartPB AND #MGB."MGB-B".IN.ReqAccessStopPB AND #MGB."MGB-B".IN.CycleStopPB AND #MGB."MGB-B".IN.StopPB);
END_REGION

REGION Network 49: **** 8 - Outputs **** Output of the Safety Gate Alarm / **** 8 - Outputs **** Output of the safety Alarm
   // Output of the Gate Alarm / Output of the Alarm
   #O_SafetyGateAlarm := #SafetyGateAlarm;
END_REGION

REGION Network 50: **** 8 - Outputs **** Output of the Safety Gate Alarm / **** 8 - Outputs **** Output of the safety Alarm / **** 8 - Outputs **** Output of the Enabling Switch Alarm
   // Output of the Gate Alarm / Output of the Alarm
   #O_EnablingSwitchAlarm := #EnablingSwitchAlarm;
END_REGION

REGION Network 51: **** 8 - Outputs **** Output of the Solenoid Alarm / **** 8 - Outputs **** Output of the Alarm
   // Output of the Solenoid Alarm / Output of the Alarm
   #O_SolenoidAlarm := #SolenoidAlarm;
END_REGION

REGION Network 52: **** 8 - Outputs **** Output of the Solenoid Alarm / **** 8 - Outputs **** Output of the Alarm / **** 8 - Outputs **** Output of the Access Request Alarm
   // Output of the Solenoid Alarm / Output of the Alarm / Output of the Access Request Alarm
   #O_AccessReqAlarm := #AccessReqAlarm;
END_REGION

REGION Network 53: **** 8 - Outputs **** Output of the MGB diagnostic warning / **** 8 - Outputs **** Output of the warning
   // Output of the MGB diagnostic warning / Output of the solenoid Alarm
   #O_MGBDiagWarning := #MGB."MGB-DIAG".IN.DiagMessagePresent OR #MGB."MGB-DIAG".IN.DiagPlausibilityCheckError OR #MGB."MGB-DIAG".IN.DiagFaultES OR #MGB."MGB-DIAG".IN.DiagFaultEnablingSw OR #MGB."MGB-DIAG".IN.DiagFaultEnablingModule;
END_REGION

REGION Network 54: **** 8 - Outputs **** Output of the alarm AB condition
   // Alarm AB condition
   #O_AlarmABCondition := #SafetyGateAlarmCond;
END_REGION

REGION Network 55: **** 8 - Outputs **** Output of the start pushbutton
   // Output of the start pushbutton
   #O_StartPB := #MGB."MGB-B".IN.StartPB;
END_REGION

REGION Network 56: **** 8 - Outputs **** Output of the reset alarm pushbutton
   // Output of the reset alarm pushbutton
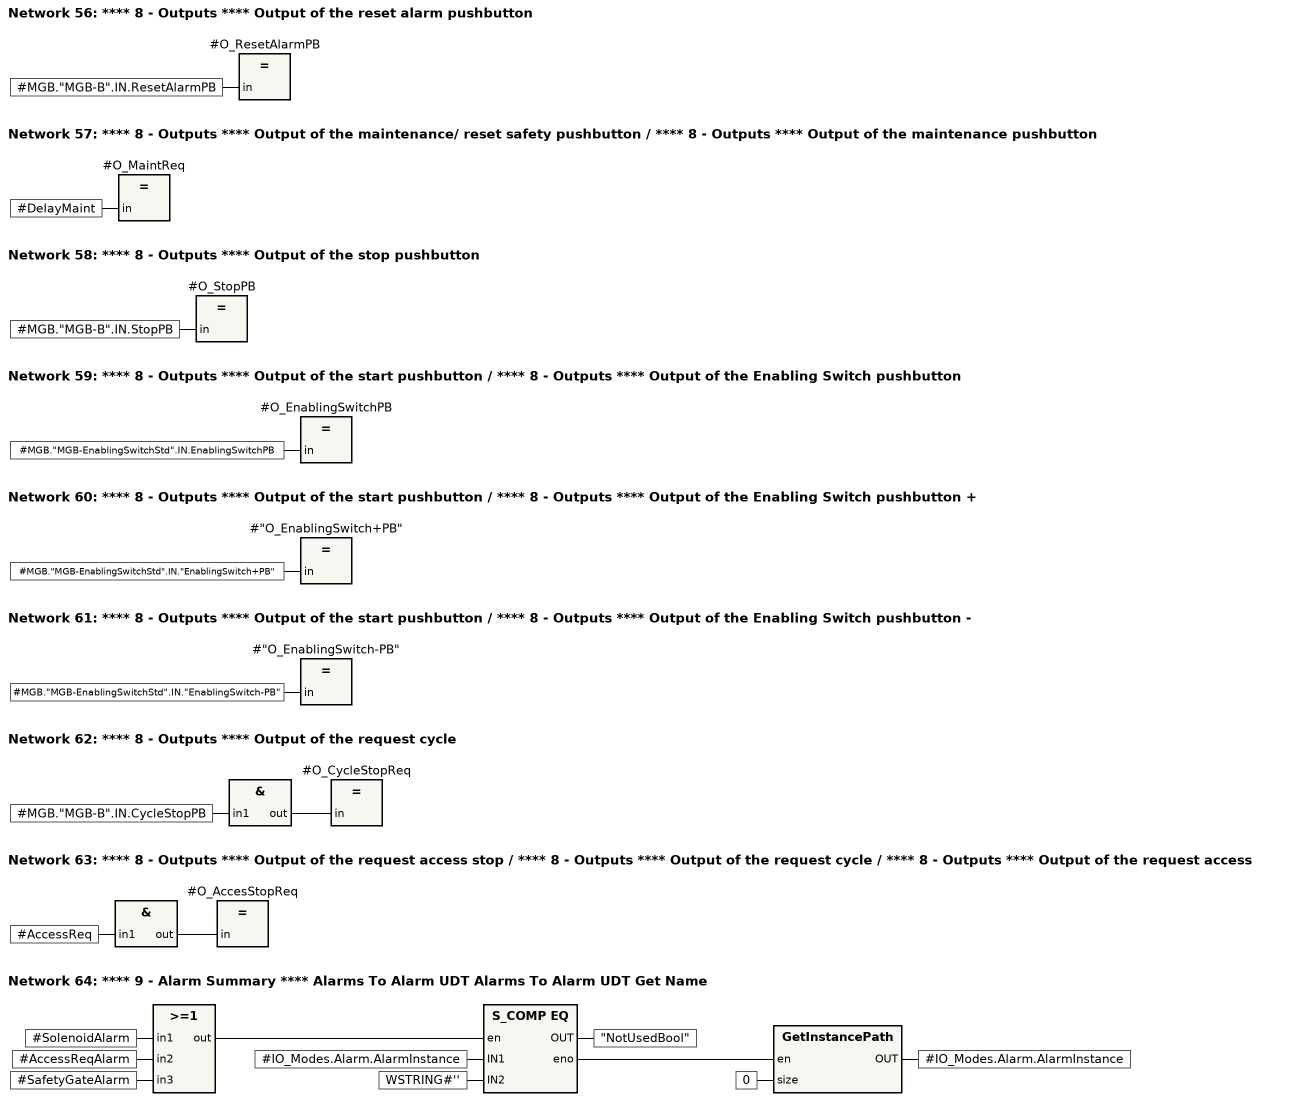
   #O_ResetAlarmPB := #MGB."MGB-B".IN.ResetAlarmPB;
END_REGION

REGION Network 57: **** 8 - Outputs **** Output of the maintenance/ reset safety pushbutton / **** 8 - Outputs **** Output of the maintenance pushbutton
   // Output of the maintenance/ reset safety pushbutton / Output of the maintenance pushbutton
   #O_MaintReq := #DelayMaint;
END_REGION

REGION Network 58: **** 8 - Outputs **** Output of the stop pushbutton
   // Output of the stop pushbutton
   #O_StopPB := #MGB."MGB-B".IN.StopPB;
END_REGION

REGION Network 59: **** 8 - Outputs **** Output of the start pushbutton / **** 8 - Outputs **** Output of the Enabling Switch pushbutton
   // Output of the start pushbutton / Output of the Enabling Switch pushbutton
   #O_EnablingSwitchPB := #MGB."MGB-EnablingSwitchStd".IN.EnablingSwitchPB;
END_REGION

REGION Network 60: **** 8 - Outputs **** Output of the start pushbutton / **** 8 - Outputs **** Output of the Enabling Switch pushbutton +
   // Output of the start pushbutton / Output of the Enabling Switch pushbutton +
   #"O_EnablingSwitch+PB" := #MGB."MGB-EnablingSwitchStd".IN."EnablingSwitch+PB";
END_REGION

REGION Network 61: **** 8 - Outputs **** Output of the start pushbutton / **** 8 - Outputs **** Output of the Enabling Switch pushbutton -
   // Output of the start pushbutton / Output of the Enabling Switch pushbutton -
   #"O_EnablingSwitch-PB" := #MGB."MGB-EnablingSwitchStd".IN."EnablingSwitch-PB";
END_REGION

REGION Network 62: **** 8 - Outputs **** Output of the request cycle
   // Output of the request cycle
   #O_CycleStopReq := #MGB."MGB-B".IN.CycleStopPB;
END_REGION

REGION Network 63: **** 8 - Outputs **** Output of the request access stop / **** 8 - Outputs **** Output of the request cycle / **** 8 - Outputs **** Output of the request access
   // Output of the request access stop / Output of the request cycle / Output of the request access
   #O_AccesStopReq := #AccessReq;
END_REGION

REGION Network 64: **** 9 - Alarm Summary **** Alarms To Alarm UDT Alarms To Alarm UDT Get Name
   // Alarm / Alarm D
   S_COMP(EN := #SolenoidAlarm OR #AccessReqAlarm OR #SafetyGateAlarm,
          IN1 := #IO_Modes.Alarm.AlarmInstance,
          IN2 := WSTRING#'',
          OUT => "NotUsedBool",
          ENO => #_w1);
   IF #_w1 THEN GetInstancePath(size := 0, OUT => #IO_Modes.Alarm.AlarmInstance); END_IF;
END_REGION

REGION Network 65: **** 9 - Alarm Summary **** Alarms To Alarm UDT
   // Alarm / Alarm D
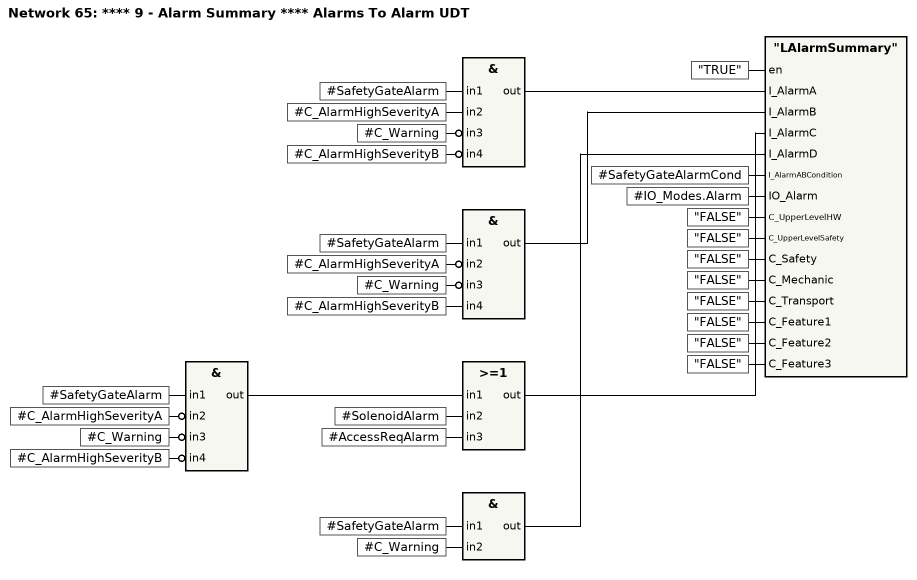
   IF "TRUE" THEN
       "LAlarmSummary"(I_AlarmA := #SafetyGateAlarm AND #C_AlarmHighSeverityA AND NOT #C_Warning AND NOT #C_AlarmHighSeverityB,
                       I_AlarmB := #SafetyGateAlarm AND NOT #C_AlarmHighSeverityA AND NOT #C_Warning AND #C_AlarmHighSeverityB,
                       I_AlarmC := (#SafetyGateAlarm AND NOT #C_AlarmHighSeverityA AND NOT #C_Warning AND NOT #C_AlarmHighSeverityB) OR #SolenoidAlarm OR #AccessReqAlarm,
                       I_AlarmD := #SafetyGateAlarm AND #C_Warning,
                       I_AlarmABCondition := #SafetyGateAlarmCond,
                       IO_Alarm := #IO_Modes.Alarm,
                       C_UpperLevelHW := "FALSE",
                       C_UpperLevelSafety := "FALSE",
                       C_Safety := "FALSE",
                       C_Mechanic := "FALSE",
                       C_Transport := "FALSE",
                       C_Feature1 := "FALSE",
                       C_Feature2 := "FALSE",
                       C_Feature3 := "FALSE");
   END_IF;
END_REGION
END_FUNCTION_BLOCK
